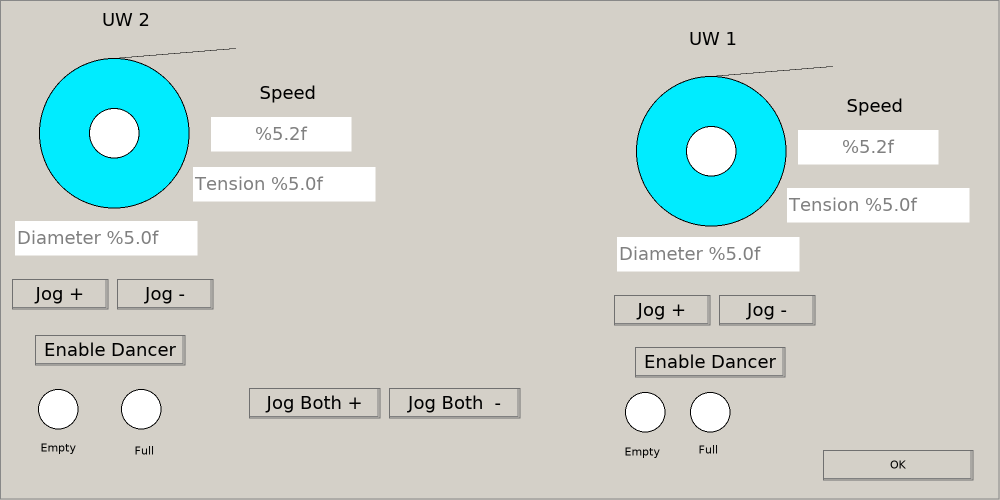
VISUALIZATION Winders  // 1000x500
    Button (823,450 150x30), "OK"
        OnMouseDown: CloseDialog Dialog=Winders, Result=OK, NumpadKeypadSet=True
    Ellipse (636,76 150x150)
    Ellipse (686,126 50x50)
    Line (698,77) (832,66)
    Ellipse (39,58 150x150)
    Ellipse (89,108 50x50)
    Line (101,59) (235,48)
    Label (638,24 150x30), "UW 1"
    Label (51,5 150x30), "UW 2"
    Textfield (616,236 184x36), "Diameter %5.0f", text variable: prg_Motion.UW_1_Diameter.Diameter_filtred
        OnMouseClick: write the text variable via Edit, min 0, max 1000000, title "Enter number of cycles"
    Button (614,295 96x30), "Jog +"
        tap gMachineCtrl.Cmd.UW_1_Cmd.JogSFwdSlow
    Button (719,295 96x30), "Jog -"
        tap gMachineCtrl.Cmd.UW_1_Cmd.JogBackdSlow
    Textfield (797,129 142x36), "%5.2f", text variable: gWebAxes.UW_1.Ref.NcToPlc.ActVelo
        OnMouseClick: write the text variable via Edit, min 0, max 1000000, title "Enter number of cycles"
    Label (800,91 150x30), "Speed"
    Textfield (210,116 142x36), "%5.2f", text variable: gWebAxes.UW_2.Ref.NcToPlc.ActVelo
        OnMouseClick: write the text variable via Edit, min 0, max 1000000, title "Enter number of cycles"
    Label (213,78 150x30), "Speed"
    Textfield (14,220 184x36), "Diameter %5.0f", text variable: prg_Motion.UW_2_Diameter.Diameter_filtred
        OnMouseClick: write the text variable via Edit, min 0, max 1000000, title "Enter number of cycles"
    Button (12,279 96x30), "Jog +"
        tap gMachineCtrl.Cmd.UW_2_Cmd.JogSFwdSlow
    Button (117,279 96x30), "Jog -"
        tap gMachineCtrl.Cmd.UW_2_Cmd.JogBackdSlow
    Button (249,388 131x30), "Jog Both +"
        OnMouseDown: execute { gMachineCtrl.Cmd.UW_2_Cmd.JogSFwdSlow := TRUE; gMachineCtrl.Cmd.UW_1_Cmd.JogSFwdSlow := TRUE; }
        OnMouseUp: execute { gMachineCtrl.Cmd.UW_2_Cmd.JogSFwdSlow := FALSE; gMachineCtrl.Cmd.UW_1_Cmd.JogSFwdSlow := FALSE; }
    Button (389,388 131x30), "Jog Both -"
        OnMouseDown: execute { gMachineCtrl.Cmd.UW_2_Cmd.JogBackdSlow := TRUE; gMachineCtrl.Cmd.UW_1_Cmd.JogBackdSlow := TRUE; }
        OnMouseUp: execute { gMachineCtrl.Cmd.UW_2_Cmd.JogBackdSlow := FALSE; gMachineCtrl.Cmd.UW_1_Cmd.JogBackdSlow := FALSE; }
    Textfield (786,187 184x36), "Tension %5.0f", text variable: prg_Motion.UW_1_Data.Tension.Tension_filtred
    Textfield (192,166 184x36), "Tension %5.0f", text variable: prg_Motion.UW_2_Data.Tension.Tension_filtred
    Button (35,335 150x30), "Enable Dancer"
        toggle gMachineCtrl.Parameters.UW_2_Param.EnableDancer
    Button (635,347 150x30), "Enable Dancer"
        toggle gMachineCtrl.Parameters.UW_1_Param.EnableDancer
    Ellipse (121,389 40x40), colour toggle: gMachineCtrl.IO.In.UW_2_DancerFull
    Ellipse (690,392 40x40), colour toggle: gMachineCtrl.IO.In.UW_1_DancerFull
    Ellipse (38,389 40x40), colour toggle: gMachineCtrl.IO.In.UW_2_DancerEmpety
    Label (27,433 63x30), "Empty"
    Label (113,436 63x30), "Full"
    Ellipse (625,392 40x40), colour toggle: gMachineCtrl.IO.In.UW_1_DancerEmpety
    Label (677,435 63x30), "Full"
    Label (611,437 63x30), "Empty"
END_VISUALIZATION

(* stored: Version 1.1.0.1, ProductVersion 3.1.4024.3
   Visu Winders: Id {00b08cf9-f7d9-4f4f-8b92-9b7903467a68} *)
